// TwinCAT 3 PLC project Panel_PC
// ProgramVersion: 3.1.4024.0
// libraries:
//   Tc2_Standard, * (Beckhoff Automation GmbH)
//   Tc2_System, * (Beckhoff Automation GmbH)
//   Tc3_Module, * (Beckhoff Automation GmbH)
// project tree:
//   DUTs/01_Enum/ E_Conveyor.TcDUT, E_MotorDOL.TcDUT, E_MotorVFD.TcDUT
//   DUTs/02_ST/ ST_Cylinder.TcDUT
//   / PlcTask.TcTTO
//   POUs/01_FB_Template/ FB_01.TcPOU, FB_02.TcPOU, FB_03.TcPOU, FB_04.TcPOU, FB_05.TcPOU, FB_06.TcPOU, FB_07.TcPOU
//   POUs/ MAIN.TcPOU
// real-time tasks:
//   TASK PlcTask: cycle T#10ms, priority 20, ADS port 350

CONFIGURATION Panel_PC
    RESOURCE PLC ON TwinCAT3
        TASK PlcTask(INTERVAL := T#10ms, PRIORITY := 20);
        PROGRAM MAIN WITH PlcTask : MAIN;
    END_RESOURCE
END_CONFIGURATION

// ---- DUTs/01_Enum/E_Conveyor.TcDUT
{attribute 'qualified_only'}
{attribute 'strict'}
TYPE E_Conveyor :
(
	enum_member := 0
);
END_TYPE

// ---- DUTs/01_Enum/E_MotorDOL.TcDUT
{attribute 'qualified_only'}
{attribute 'strict'}
TYPE E_MotorDOL :
(
	enum_member := 0
);
END_TYPE

// ---- DUTs/01_Enum/E_MotorVFD.TcDUT
{attribute 'qualified_only'}
{attribute 'strict'}
TYPE E_MotorVFD :
(
	enum_member := 0
);
END_TYPE

// ---- DUTs/02_ST/ST_Cylinder.TcDUT
TYPE ST_Cylinder :
STRUCT
END_STRUCT
END_TYPE

// ---- POUs/MAIN.TcPOU
PROGRAM MAIN
VAR
END_VAR

END_PROGRAM

// ---- POUs/01_FB_Template/FB_01.TcPOU
FUNCTION_BLOCK FB_01
VAR_INPUT
END_VAR
VAR_OUTPUT
END_VAR
VAR
END_VAR

END_FUNCTION_BLOCK

// ---- POUs/01_FB_Template/FB_02.TcPOU
FUNCTION_BLOCK FB_02
VAR_INPUT
END_VAR
VAR_OUTPUT
END_VAR
VAR
END_VAR

END_FUNCTION_BLOCK

// ---- POUs/01_FB_Template/FB_03.TcPOU
FUNCTION_BLOCK FB_03
VAR_INPUT
END_VAR
VAR_OUTPUT
END_VAR
VAR
END_VAR

END_FUNCTION_BLOCK

// ---- POUs/01_FB_Template/FB_04.TcPOU
FUNCTION_BLOCK FB_04
VAR_INPUT
END_VAR
VAR_OUTPUT
END_VAR
VAR
END_VAR

END_FUNCTION_BLOCK

// ---- POUs/01_FB_Template/FB_05.TcPOU
FUNCTION_BLOCK FB_05
VAR_INPUT
END_VAR
VAR_OUTPUT
END_VAR
VAR
END_VAR

END_FUNCTION_BLOCK

// ---- POUs/01_FB_Template/FB_06.TcPOU
FUNCTION_BLOCK FB_06
VAR_INPUT
	Trong AT %I* : BOOL;
END_VAR
VAR_OUTPUT
END_VAR
VAR
END_VAR

END_FUNCTION_BLOCK

// ---- POUs/01_FB_Template/FB_07.TcPOU
FUNCTION_BLOCK FB_07
VAR_INPUT
	TRONG AT %I* : BOOL;
END_VAR
VAR_OUTPUT
END_VAR
VAR
END_VAR

END_FUNCTION_BLOCK
